FUNCTION_BLOCK FB_500_VG
VAR_IN_OUT
	IG : ST_VG;
END_VAR
VAR_INPUT
	PG	:	ST_VG;
END_VAR
VAR_OUTPUT
	xHV_SW: BOOL;
	rPRESS: INT;
	rVAC_SP: INT;
END_VAR
VAR
	rV : REAL;
	GaugeTurnOnTmr : TON;
	MinPressure: REAL := 1E-9;
	
END_VAR
VAR CONSTANT
	cDefaultPressure : REAL := 750.0;
	vBase	:	REAL := 1; //corresponding vbase 1V actually?
	pBase	:	REAL := 1.0E-9; //i think the pbase might be 1E-9 for the default curve...
	vSlope	:	REAL := 1.0; //looks correct for default curve
END_VAR

(* 500 Logarithmic Output Conversion, factory default configuration *)

rV := 10*INT_TO_REAL(IG.iPRESS_R)/32767;

IF rV >= 0.5 AND rV < 1.0  THEN
	IG.wState := 5;
	IG.rPRESS := cDefaultPressure;
ELSIF rV < 0.4 THEN
	IG.wState := 4;//HV Off/ gauge disconnected
	IG.rPRESS := cDefaultPressure;
ELSE
	IG.wState := 1;
	IG.rPRESS := EXPT(10,((rV-vBase)/vSlope+LOG(pBase)));
END_IF



(* Ion Gauge Protection Functions *)
(* If the PG pressure is greater than the VG.PRO_SP then the gauge is disabled *)
(* If the PG pressure is less than the VG.PRO_SP then the gauge is enabled *)
(* This FB also implements some hysteresis so the gauge doesn't have rapid power cycling while near the turn on boundary *)



IF PG.rPRESS < IG.rPRO_SP AND PG.xPRESS_OK THEN

	IG.xHV_DIS := IG.xHV_SW;

ELSIF IG.xHV_DIS THEN
	IF IG.rPRESS > (IG.rPRO_SP + IG.rHYS_PR)  OR PG.rPRESS > (IG.rPRO_SP + IG.rHYS_PR) THEN
		IG.xHV_DIS := FALSE;
		IG.xHV_SW := FALSE;
	END_IF
ELSE
	IG.xHV_DIS := FALSE;
	IG.xHV_SW := FALSE;
END_IF

(* Pressure gauge OK checks *)

//Backwards compatibility
IG.xPRESS_OK := (IG.wState = 1) OR IG.xBAKEOUT;

(* Setpoint evaluation *)
IG.xAT_VAC := (IG.xPRESS_OK AND (IG.rPRESS < IG.rVAC_SP)) OR IG.xBAKEOUT;;

END_FUNCTION_BLOCK

(* stored: Version 1.1.0.1, ProductVersion 3.1.4018.5
   POU FB_500_VG: Id {6241046a-c3ba-40b6-8b76-514cf5cc9cb4}, SpecialFunc None *)
